Fanuc KAREL source: kb00037.KL

PROGRAM KB00037
%STACKSIZE=65535
%PRIORITY=65535
%NOLOCKGROUP
VAR
P1 : REAL
P2 : INTEGER
P3 : INTEGER
P4 : STRING[80]
BEGIN
P1=1.0
P2=1
P3=1
P4='A'
CNV_REAL_STR(P1,P2,P3,P4)
END KB00037
